Staubli VAL3: CIRCLE.dtx

public num distance
public num moveType = 1
public num nArmType
public num nArray = 1
public num nCenterSpeed = 100
public num nCurveIn = 0.5
public num nCurveOut = 0.5
public num nCutIn = 0.5
public num nCutInOutBlend = 0.05
public num nCutOut = 0.5
public num nFrameIndex = 1
public num nGasPressure = 90
public num nIndexGun = 1
public num nJointSpeed = 100
public num nLaserDelay = 0.5
public num nLaserPower = 60
public num nOverPass
public num nPointQuantity = 1000
public num nRadius = 10
public num nStop
public num nTcpAction[9] = 1
public num nTime
public num nTotalPoint
public num nX
public num nXlength
public num nXoffset
public num nY
public num nYlength
public num nYoffset
public num nPWMPercent = 100
public num nOpenAngle
public num nJointMode
public string comment = "cicle..."
public string instruction[9]
public string sAction[3]
public bool bCutting
public bool bRes
public bool toStop
public frame fTrack = {x=34, fatherId=world[0]}
public jointRx jConfig
public jointRx jReadyIn
public jointRx jReadyOut
public jointRx jSynJoint[10]
public pointRx pCenter = {fatherId=fTrack[0]}
public pointRx pCutting[11]
  [0] = {fatherId=fTrack[0]}
  [1] = {fatherId=fTrack[0]}
  [2] = {fatherId=fTrack[0]}
  [3] = {fatherId=fTrack[0]}
  [4] = {fatherId=fTrack[0]}
  [5] = {fatherId=fTrack[0]}
  [6] = {fatherId=fTrack[0]}
  [7] = {fatherId=fTrack[0]}
  [8] = {fatherId=fTrack[0]}
  [9] = {fatherId=fTrack[0]}
  [10] = {fatherId=fTrack[0]}
public pointRx pMoveTo = {fatherId=fTrack[0]}
public pointRx pO = {fatherId=world[0]}
public pointRx pX = {fatherId=world[0]}
public pointRx pY = {fatherId=world[0]}
public pointRx points = {wrist=wfree, fatherId=fTrack[0]}
public mdesc nom_speed = {tmax=66.66, rmax=60, leave=0.05, reach=0.05}
public mdesc mJointSpeed = {vel=50, tmax=9999, rmax=9999, leave=30, reach=30}
